{attribute addProperty BoxType "EJ1914-0000-0017"}
{attribute addProperty Id "FIELDVOLTAGE_Field_Voltage_StatusFIELDVOLTAGE_Field_Voltage_Status_CAC01FE2162"}
{attribute addProperty CRC "4213925847"}
{attribute addProperty SizeInBites "16"}
{attribute addProperty SizeInBytes "2"}
TYPE Module_2_DEVICEIO_FB2B67D7 :
STRUCT
	{attribute addProperty Name "FIELDVOLTAGE_Field_Voltage_Status"}
	FIELDVOLTAGE_Field_Voltage_Status  : FIELDVOLTAGE_Field_Voltage_Status_CAC01FE2;
END_STRUCT
END_TYPE

(* stored: Version 1.2.0.0, ProductVersion 3.1.4024.9
   DUT Module_2_DEVICEIO_FB2B67D7: Id {60a3ce8d-646a-4e39-91e3-85796411115d} *)
